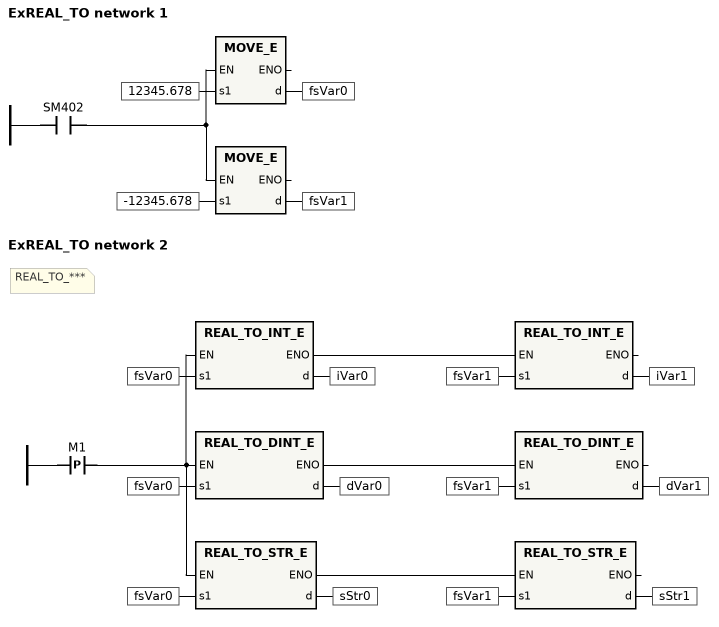
(* [picture p24: structured ladder/FBD of ExREAL_TO, networks 1 to 2] *)
(* network 1 *)
MOVE_E(SM402, 12345.678, fsVar0);
MOVE_E(SM402, -12345.678, fsVar1);
(* network 2 *)
(* REAL_TO_*** *)
_p1 := LDP(TRUE, M1);
_e2 := REAL_TO_INT_E(_p1, fsVar0, iVar0);
REAL_TO_INT_E(_e2, fsVar1, iVar1);
_e3 := REAL_TO_DINT_E(_p1, fsVar0, dVar0);
REAL_TO_DINT_E(_e3, fsVar1, dVar1);
_e4 := REAL_TO_STR_E(_p1, fsVar0, sStr0);
REAL_TO_STR_E(_e4, fsVar1, sStr1);
END_PROGRAM

PROGRAM ExSTR_TO
VAR
  GetInt : INT;
  NthBit : INT;
  SetInt : INT;
  SetInt2 : INT;
END_VAR
(* structured ladder/FBD written out as ST: instructions are called as NAME(EN, inputs, outputs); _pN, _eN, _tN stand for wires *)
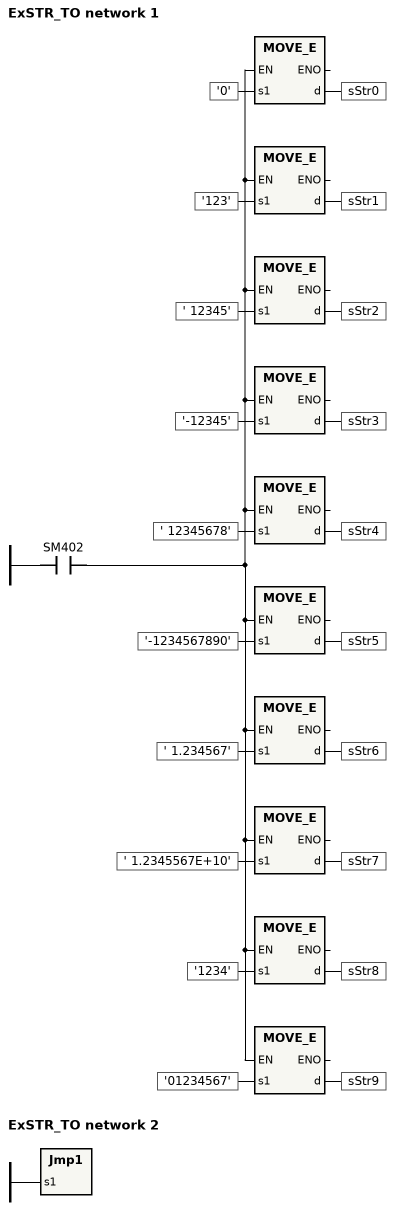
(* network 1 *)
MOVE_E(SM402, '0', sStr0);
MOVE_E(SM402, '123', sStr1);
MOVE_E(SM402, ' 12345', sStr2);
MOVE_E(SM402, '-12345', sStr3);
MOVE_E(SM402, ' 12345678', sStr4);
MOVE_E(SM402, '-1234567890', sStr5);
MOVE_E(SM402, ' 1.234567', sStr6);
MOVE_E(SM402, ' 1.2345567E+10', sStr7);
MOVE_E(SM402, '1234', sStr8);
MOVE_E(SM402, '01234567', sStr9);
(* network 2 *)
(* element kind 9 Jmp1 <- TRUE *)
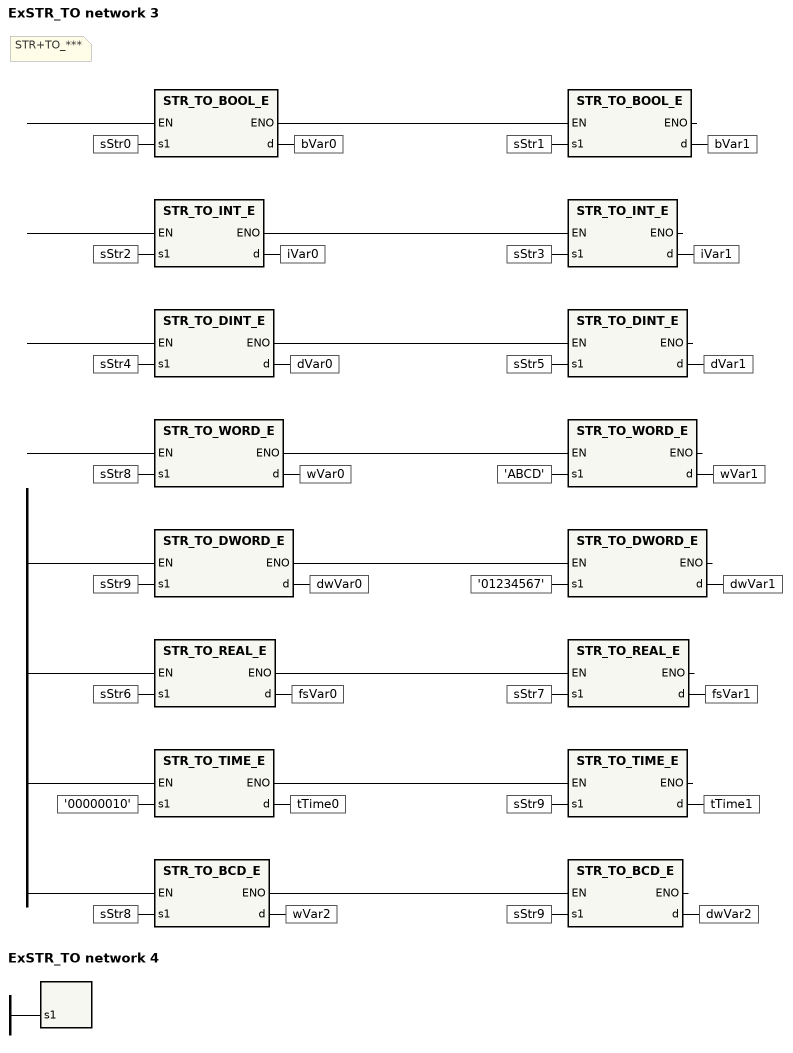
(* network 3 *)
(* STR+TO_*** *)
_e1 := STR_TO_BOOL_E(TRUE, sStr0, bVar0);
STR_TO_BOOL_E(_e1, sStr1, bVar1);
_e2 := STR_TO_INT_E(TRUE, sStr2, iVar0);
STR_TO_INT_E(_e2, sStr3, iVar1);
_e3 := STR_TO_DINT_E(TRUE, sStr4, dVar0);
STR_TO_DINT_E(_e3, sStr5, dVar1);
_e4 := STR_TO_WORD_E(TRUE, sStr8, wVar0);
STR_TO_WORD_E(_e4, 'ABCD', wVar1);
_e5 := STR_TO_DWORD_E(TRUE, sStr9, dwVar0);
STR_TO_DWORD_E(_e5, '01234567', dwVar1);
_e6 := STR_TO_REAL_E(TRUE, sStr6, fsVar0);
STR_TO_REAL_E(_e6, sStr7, fsVar1);
_e7 := STR_TO_TIME_E(TRUE, '00000010', tTime0);
STR_TO_TIME_E(_e7, sStr9, tTime1);
_e8 := STR_TO_BCD_E(TRUE, sStr8, wVar2);
STR_TO_BCD_E(_e8, sStr9, dwVar2);
(* network 4 *)
(* element kind 10  <- TRUE *)
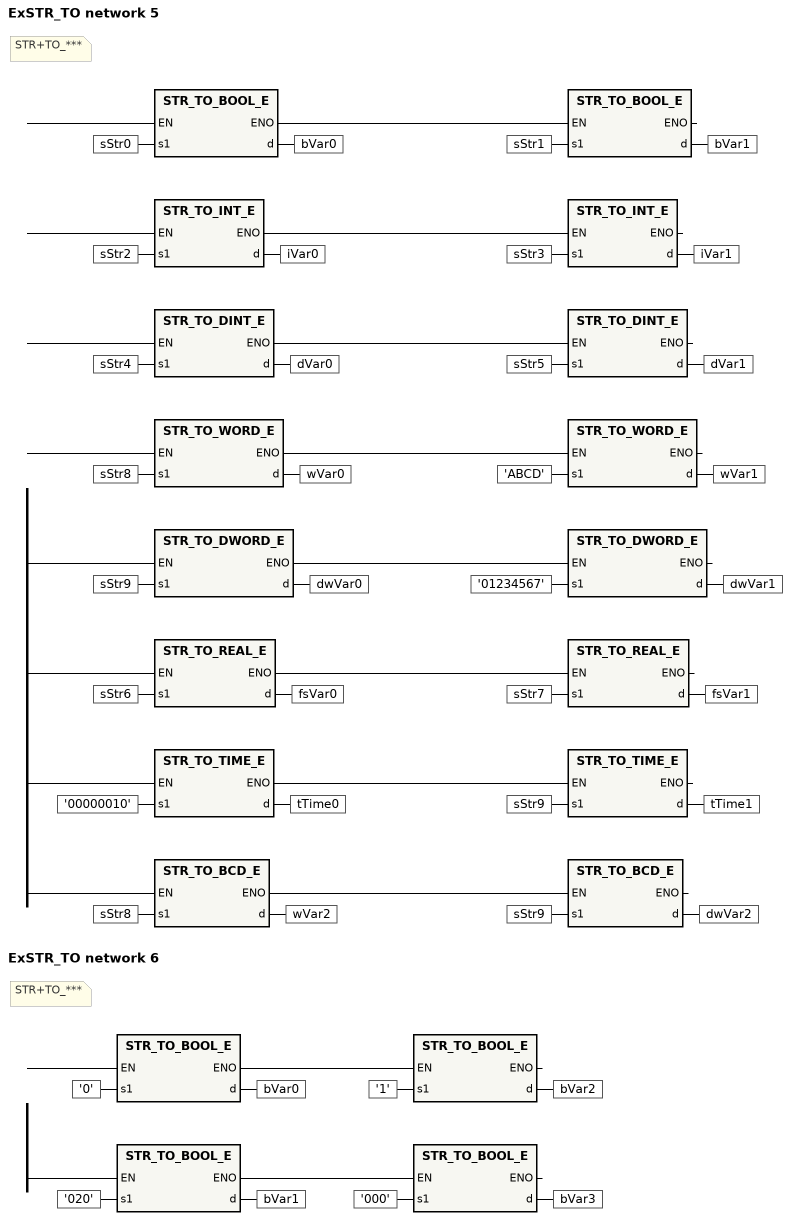
(* network 5 *)
(* STR+TO_*** *)
_e1 := STR_TO_BOOL_E(TRUE, sStr0, bVar0);
STR_TO_BOOL_E(_e1, sStr1, bVar1);
_e2 := STR_TO_INT_E(TRUE, sStr2, iVar0);
STR_TO_INT_E(_e2, sStr3, iVar1);
_e3 := STR_TO_DINT_E(TRUE, sStr4, dVar0);
STR_TO_DINT_E(_e3, sStr5, dVar1);
_e4 := STR_TO_WORD_E(TRUE, sStr8, wVar0);
STR_TO_WORD_E(_e4, 'ABCD', wVar1);
_e5 := STR_TO_DWORD_E(TRUE, sStr9, dwVar0);
STR_TO_DWORD_E(_e5, '01234567', dwVar1);
_e6 := STR_TO_REAL_E(TRUE, sStr6, fsVar0);
STR_TO_REAL_E(_e6, sStr7, fsVar1);
_e7 := STR_TO_TIME_E(TRUE, '00000010', tTime0);
STR_TO_TIME_E(_e7, sStr9, tTime1);
_e8 := STR_TO_BCD_E(TRUE, sStr8, wVar2);
STR_TO_BCD_E(_e8, sStr9, dwVar2);
(* network 6 Jmp1: *)
(* STR+TO_*** *)
_e1 := STR_TO_BOOL_E(TRUE, '0', bVar0);
STR_TO_BOOL_E(_e1, '1', bVar2);
_e2 := STR_TO_BOOL_E(TRUE, '020', bVar1);
STR_TO_BOOL_E(_e2, '000', bVar3);
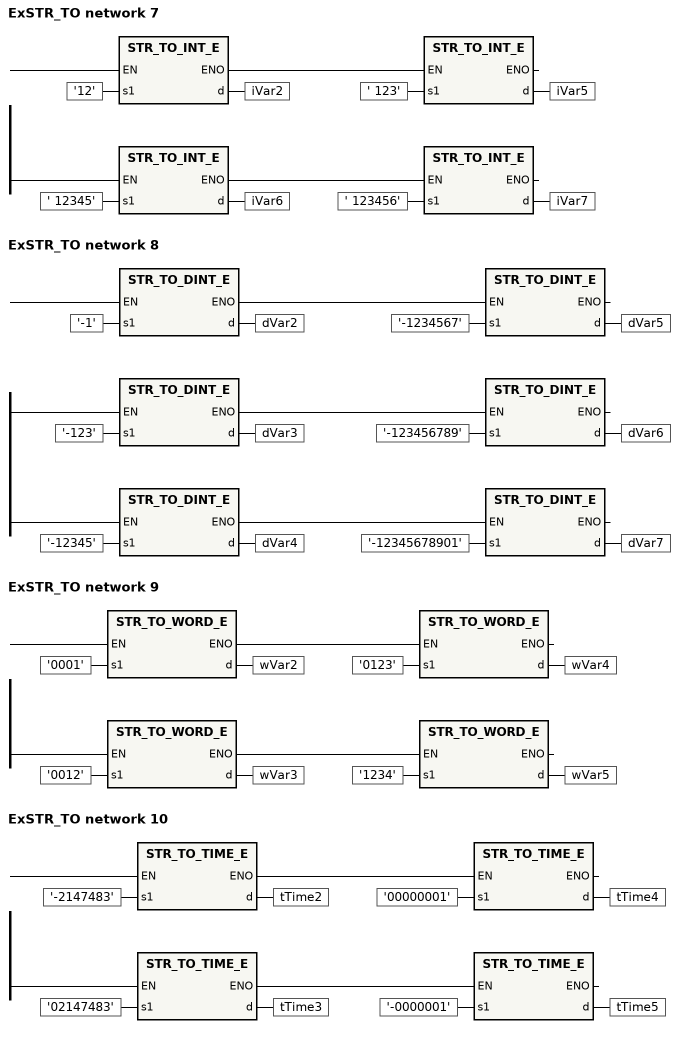
(* network 7 *)
_e1 := STR_TO_INT_E(TRUE, '12', iVar2);
STR_TO_INT_E(_e1, ' 123', iVar5);
_e2 := STR_TO_INT_E(TRUE, ' 12345', iVar6);
STR_TO_INT_E(_e2, ' 123456', iVar7);
(* network 8 *)
_e1 := STR_TO_DINT_E(TRUE, '-1', dVar2);
STR_TO_DINT_E(_e1, '-1234567', dVar5);
_e2 := STR_TO_DINT_E(TRUE, '-123', dVar3);
STR_TO_DINT_E(_e2, '-123456789', dVar6);
_e3 := STR_TO_DINT_E(TRUE, '-12345', dVar4);
STR_TO_DINT_E(_e3, '-12345678901', dVar7);
(* network 9 *)
_e1 := STR_TO_WORD_E(TRUE, '0001', wVar2);
STR_TO_WORD_E(_e1, '0123', wVar4);
_e2 := STR_TO_WORD_E(TRUE, '0012', wVar3);
STR_TO_WORD_E(_e2, '1234', wVar5);
(* network 10 *)
_e1 := STR_TO_TIME_E(TRUE, '-2147483', tTime2);
STR_TO_TIME_E(_e1, '00000001', tTime4);
_e2 := STR_TO_TIME_E(TRUE, '02147483', tTime3);
STR_TO_TIME_E(_e2, '-0000001', tTime5);
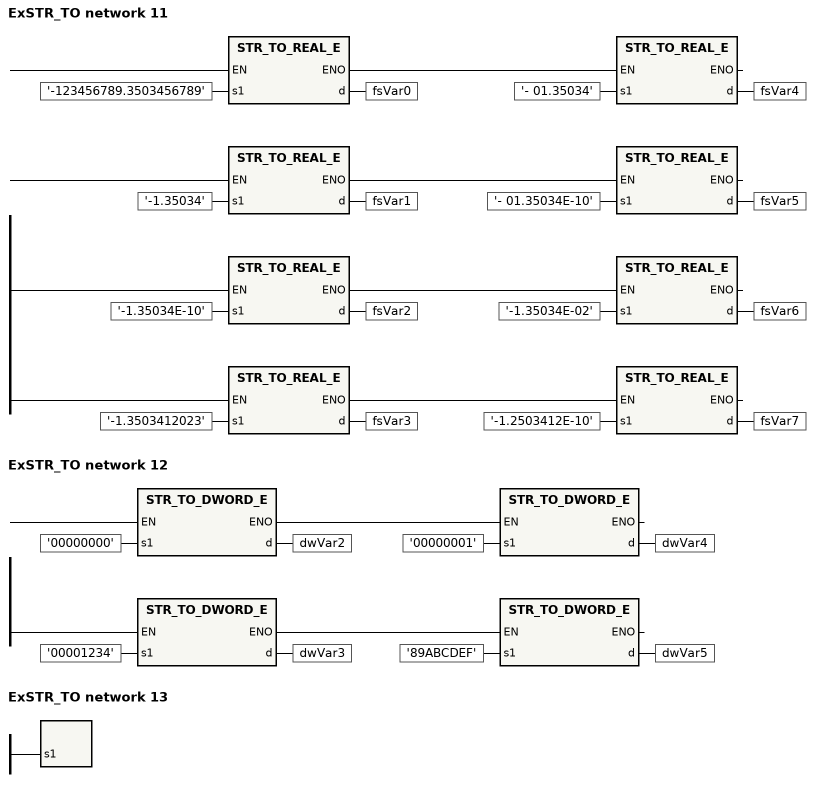
(* network 11 *)
_e1 := STR_TO_REAL_E(TRUE, '-123456789.3503456789', fsVar0);
STR_TO_REAL_E(_e1, '- 01.35034', fsVar4);
_e2 := STR_TO_REAL_E(TRUE, '-1.35034', fsVar1);
STR_TO_REAL_E(_e2, '- 01.35034E-10', fsVar5);
_e3 := STR_TO_REAL_E(TRUE, '-1.35034E-10', fsVar2);
STR_TO_REAL_E(_e3, '-1.35034E-02', fsVar6);
_e4 := STR_TO_REAL_E(TRUE, '-1.3503412023', fsVar3);
STR_TO_REAL_E(_e4, '-1.2503412E-10', fsVar7);
(* network 12 *)
_e1 := STR_TO_DWORD_E(TRUE, '00000000', dwVar2);
STR_TO_DWORD_E(_e1, '00000001', dwVar4);
_e2 := STR_TO_DWORD_E(TRUE, '00001234', dwVar3);
STR_TO_DWORD_E(_e2, '89ABCDEF', dwVar5);
(* network 13 *)
(* element kind 10  <- TRUE *)
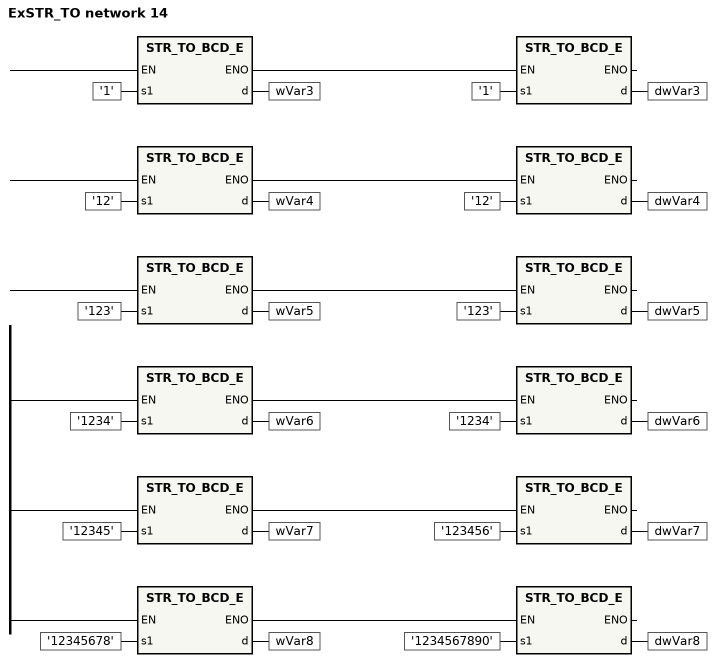
(* network 14 Jmp2: *)
_e1 := STR_TO_BCD_E(TRUE, '1', wVar3);
STR_TO_BCD_E(_e1, '1', dwVar3);
_e2 := STR_TO_BCD_E(TRUE, '12', wVar4);
STR_TO_BCD_E(_e2, '12', dwVar4);
_e3 := STR_TO_BCD_E(TRUE, '123', wVar5);
STR_TO_BCD_E(_e3, '123', dwVar5);
_e4 := STR_TO_BCD_E(TRUE, '1234', wVar6);
STR_TO_BCD_E(_e4, '1234', dwVar6);
_e5 := STR_TO_BCD_E(TRUE, '12345', wVar7);
STR_TO_BCD_E(_e5, '123456', dwVar7);
_e6 := STR_TO_BCD_E(TRUE, '12345678', wVar8);
STR_TO_BCD_E(_e6, '1234567890', dwVar8);
END_PROGRAM

PROGRAM ExTIME_TO
VAR
  GetInt : INT;
  NthBit : INT;
  SetInt : INT;
  SetInt2 : INT;
END_VAR
(* structured ladder/FBD written out as ST: instructions are called as NAME(EN, inputs, outputs); _pN, _eN, _tN stand for wires *)
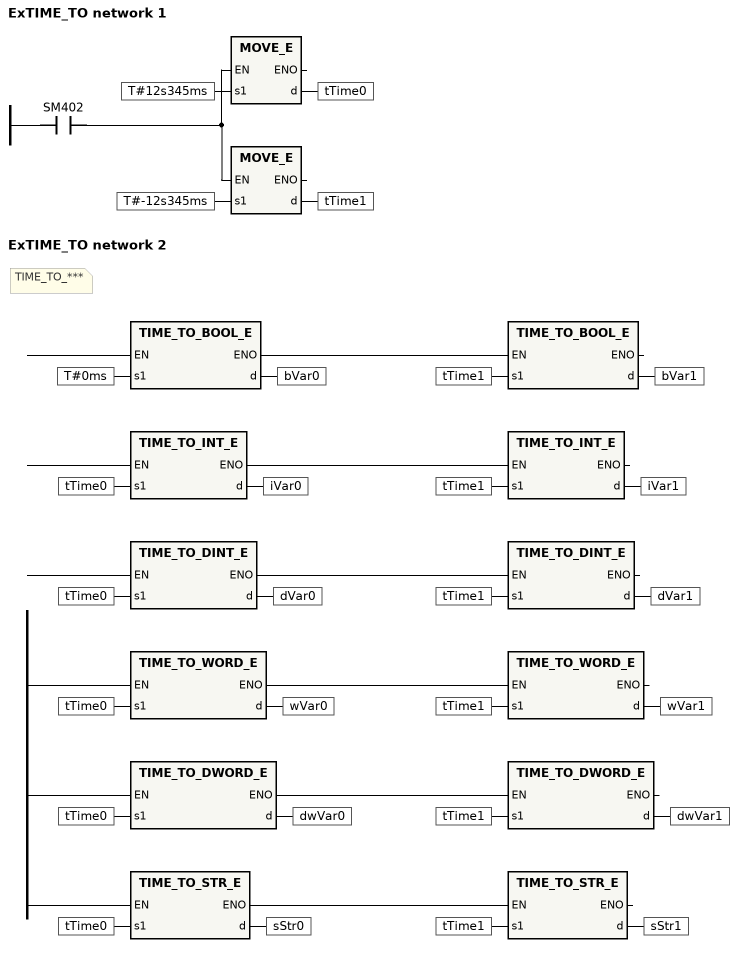
(* network 1 *)
MOVE_E(SM402, T#12s345ms, tTime0);
MOVE_E(SM402, T#-12s345ms, tTime1);
(* network 2 *)
(* TIME_TO_*** *)
_e1 := TIME_TO_BOOL_E(TRUE, T#0ms, bVar0);
TIME_TO_BOOL_E(_e1, tTime1, bVar1);
_e2 := TIME_TO_INT_E(TRUE, tTime0, iVar0);
TIME_TO_INT_E(_e2, tTime1, iVar1);
_e3 := TIME_TO_DINT_E(TRUE, tTime0, dVar0);
TIME_TO_DINT_E(_e3, tTime1, dVar1);
_e4 := TIME_TO_WORD_E(TRUE, tTime0, wVar0);
TIME_TO_WORD_E(_e4, tTime1, wVar1);
_e5 := TIME_TO_DWORD_E(TRUE, tTime0, dwVar0);
TIME_TO_DWORD_E(_e5, tTime1, dwVar1);
_e6 := TIME_TO_STR_E(TRUE, tTime0, sStr0);
TIME_TO_STR_E(_e6, tTime1, sStr1);
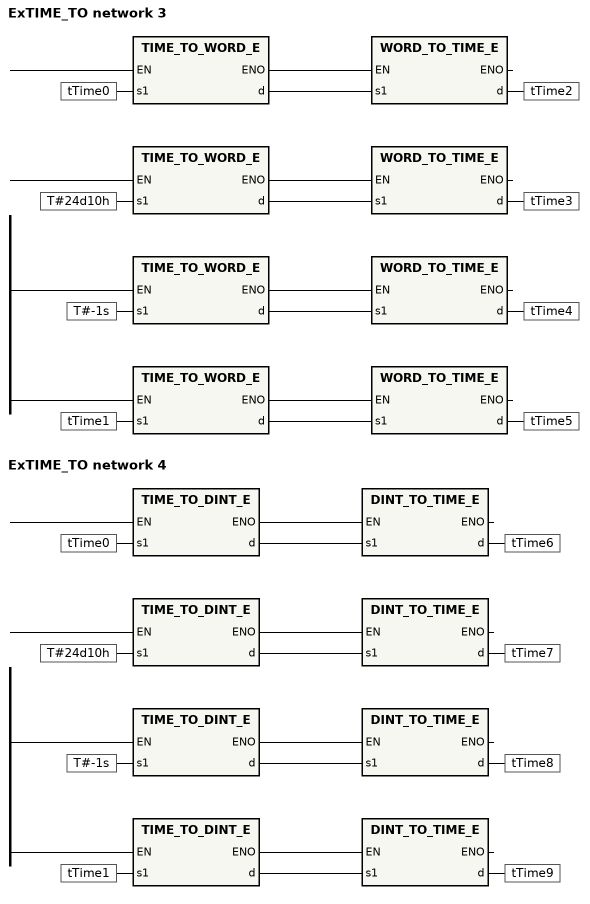
(* network 3 *)
_e2 := TIME_TO_WORD_E(TRUE, tTime0, _t1);
WORD_TO_TIME_E(_e2, _t1, tTime2);
_e4 := TIME_TO_WORD_E(TRUE, T#24d10h, _t3);
WORD_TO_TIME_E(_e4, _t3, tTime3);
_e6 := TIME_TO_WORD_E(TRUE, T#-1s, _t5);
WORD_TO_TIME_E(_e6, _t5, tTime4);
_e8 := TIME_TO_WORD_E(TRUE, tTime1, _t7);
WORD_TO_TIME_E(_e8, _t7, tTime5);
(* network 4 *)
_e2 := TIME_TO_DINT_E(TRUE, tTime0, _t1);
DINT_TO_TIME_E(_e2, _t1, tTime6);
_e4 := TIME_TO_DINT_E(TRUE, T#24d10h, _t3);
DINT_TO_TIME_E(_e4, _t3, tTime7);
_e6 := TIME_TO_DINT_E(TRUE, T#-1s, _t5);
DINT_TO_TIME_E(_e6, _t5, tTime8);
_e8 := TIME_TO_DINT_E(TRUE, tTime1, _t7);
DINT_TO_TIME_E(_e8, _t7, tTime9);
END_PROGRAM

PROGRAM ExWORD_TO
VAR
  GetInt : INT;
  NthBit : INT;
  SetInt : INT;
  SetInt2 : INT;
END_VAR
(* structured ladder/FBD written out as ST: instructions are called as NAME(EN, inputs, outputs); _pN, _eN, _tN stand for wires *)
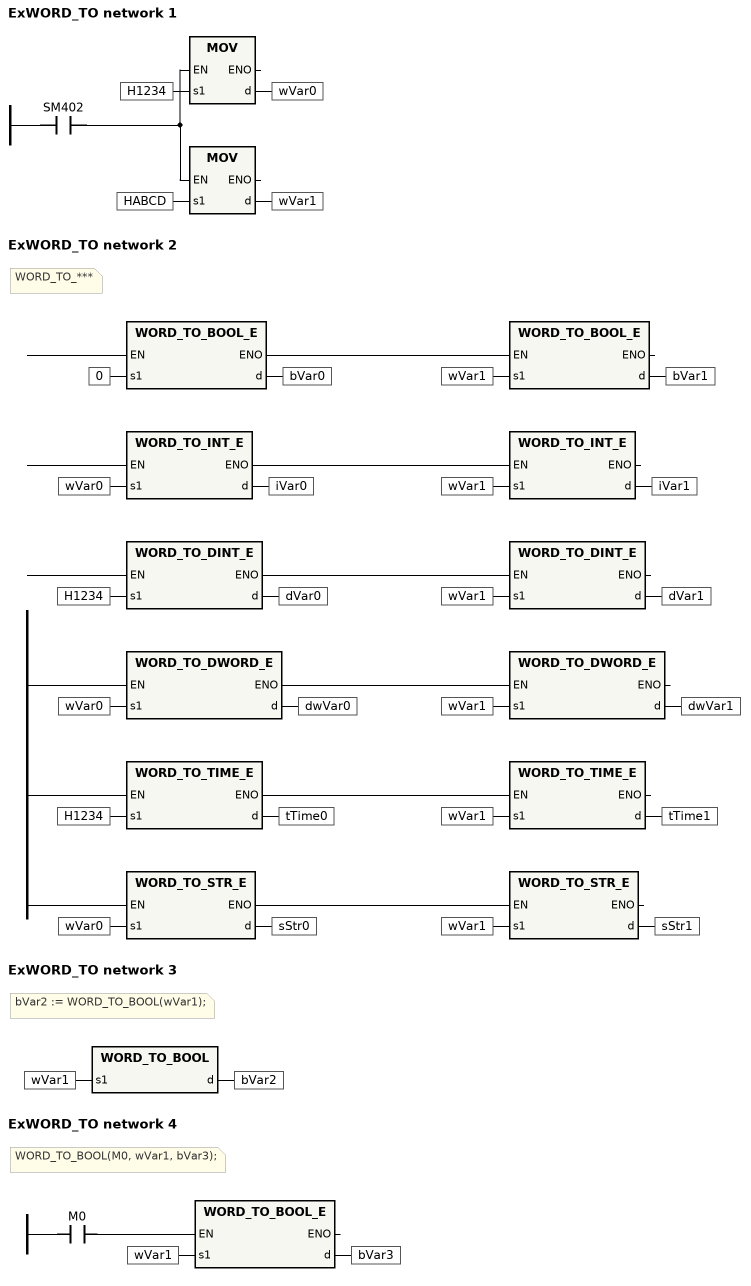
(* network 1 *)
MOV(SM402, H1234, wVar0);
MOV(SM402, HABCD, wVar1);
(* network 2 *)
(* WORD_TO_*** *)
_e1 := WORD_TO_BOOL_E(TRUE, 0, bVar0);
WORD_TO_BOOL_E(_e1, wVar1, bVar1);
_e2 := WORD_TO_INT_E(TRUE, wVar0, iVar0);
WORD_TO_INT_E(_e2, wVar1, iVar1);
_e3 := WORD_TO_DINT_E(TRUE, H1234, dVar0);
WORD_TO_DINT_E(_e3, wVar1, dVar1);
_e4 := WORD_TO_DWORD_E(TRUE, wVar0, dwVar0);
WORD_TO_DWORD_E(_e4, wVar1, dwVar1);
_e5 := WORD_TO_TIME_E(TRUE, H1234, tTime0);
WORD_TO_TIME_E(_e5, wVar1, tTime1);
_e6 := WORD_TO_STR_E(TRUE, wVar0, sStr0);
WORD_TO_STR_E(_e6, wVar1, sStr1);
(* network 3 *)
(* bVar2 := WORD_TO_BOOL(wVar1); *)
bVar2 := WORD_TO_BOOL(wVar1);
(* network 4 *)
(* WORD_TO_BOOL(M0, wVar1, bVar3); *)
WORD_TO_BOOL_E(M0, wVar1, bVar3);
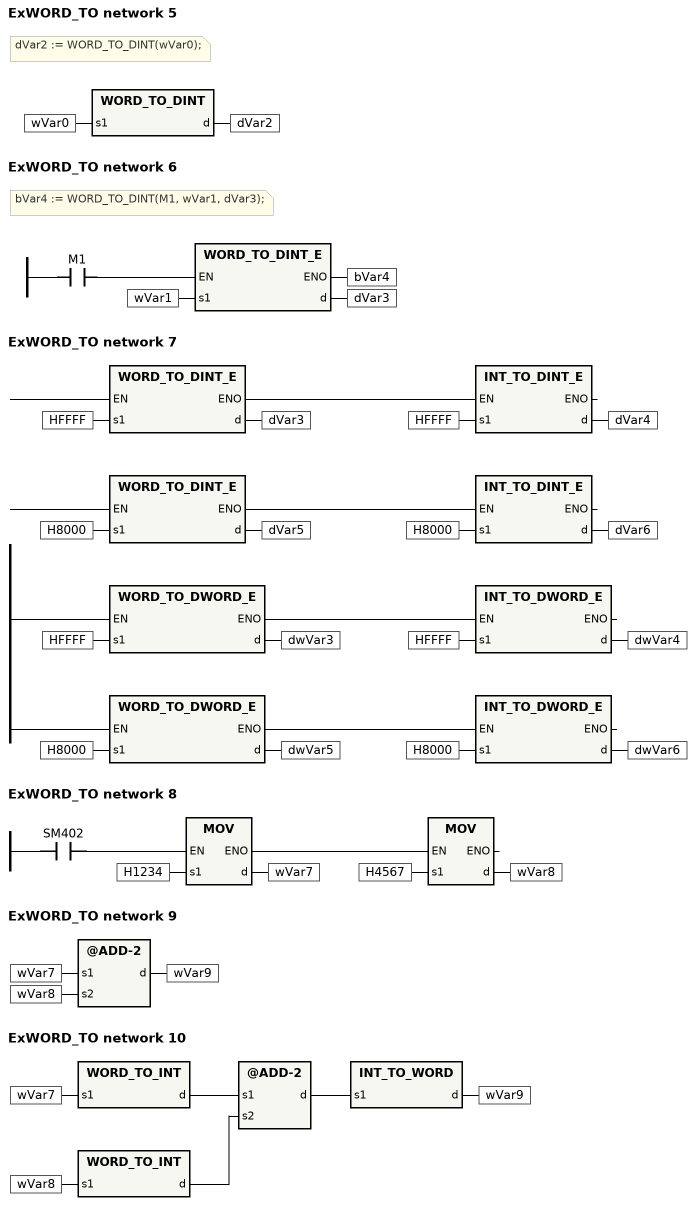
(* network 5 *)
(* dVar2 := WORD_TO_DINT(wVar0); *)
dVar2 := WORD_TO_DINT(wVar0);
(* network 6 *)
(* bVar4 := WORD_TO_DINT(M1, wVar1, dVar3); *)
_e1 := WORD_TO_DINT_E(M1, wVar1, dVar3);
bVar4 := _e1;
(* network 7 *)
_e1 := WORD_TO_DINT_E(TRUE, HFFFF, dVar3);
INT_TO_DINT_E(_e1, HFFFF, dVar4);
_e2 := WORD_TO_DINT_E(TRUE, H8000, dVar5);
INT_TO_DINT_E(_e2, H8000, dVar6);
_e3 := WORD_TO_DWORD_E(TRUE, HFFFF, dwVar3);
INT_TO_DWORD_E(_e3, HFFFF, dwVar4);
_e4 := WORD_TO_DWORD_E(TRUE, H8000, dwVar5);
INT_TO_DWORD_E(_e4, H8000, dwVar6);
(* network 8 *)
_e1 := MOV(SM402, H1234, wVar7);
MOV(_e1, H4567, wVar8);
(* network 9 *)
wVar9 := @ADD-2(wVar7, wVar8);
(* network 10 *)
wVar9 := INT_TO_WORD(@ADD-2(WORD_TO_INT(wVar7), WORD_TO_INT(wVar8)));
END_PROGRAM

FUNCTION_BLOCK INT2Bit
VAR_INPUT
  IN : INT;
END_VAR
VAR_OUTPUT
  Bit0 : BOOL;
  Bit1 : BOOL;
  Bit2 : BOOL;
  Bit3 : BOOL;
  Bit4 : BOOL;
  Bit5 : BOOL;
  Bit6 : BOOL;
  Bit7 : BOOL;
  Bit8 : BOOL;
  Bit9 : BOOL;
  Bit10 : BOOL;
  Bit11 : BOOL;
  Bit12 : BOOL;
  Bit13 : BOOL;
  Bit14 : BOOL;
  Bit15 : BOOL;
END_VAR
VAR
  abArr16 : ARRAY [0..15] OF BOOL;
END_VAR
 
abArr16[0] := INT_TO_BITARR(IN, 16);
Bit0 := abArr16[0];
Bit1 := abArr16[1];
Bit2 := abArr16[2];
Bit3 := abArr16[3];
Bit4 := abArr16[4];
Bit5 := abArr16[5];
Bit6 := abArr16[6];
Bit7 := abArr16[7];
Bit8 := abArr16[8];
Bit9 := abArr16[9];
Bit10 := abArr16[10];
Bit11 := abArr16[11];
Bit12 := abArr16[12];
Bit13 := abArr16[13];
Bit14 := abArr16[14];
Bit15 := abArr16[15];
END_FUNCTION_BLOCK

PROGRAM ExBCD_TO2
VAR
  aTank : ARRAY [0..31] OF INT;
  awStatus : ARRAY [0..9] OF WORD;
  asName : ARRAY [0..4] OF STRING[32] := [5('')];
  atDelay : ARRAY [0..4] OF TIME := [5(T#0s)];
  HMI20_1 : HMI20;
  Mov4WORD_1 : Mov4WORD;
  Mov4DWORD_1 : Mov4DWORD;
END_VAR
(* structured ladder/FBD written out as ST: instructions are called as NAME(EN, inputs, outputs); _pN, _eN, _tN stand for wires *)
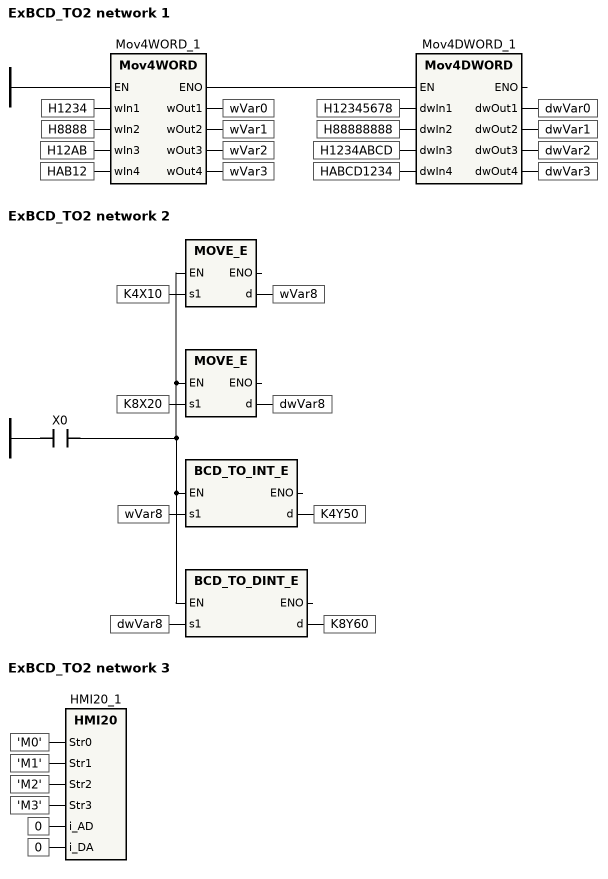
(* network 1 *)
Mov4WORD_1(EN := TRUE, wIn1 := H1234, wIn2 := H8888, wIn3 := H12AB, wIn4 := HAB12, wOut1 => wVar0, wOut2 => wVar1, wOut3 => wVar2, wOut4 => wVar3);
Mov4DWORD_1(EN := Mov4WORD_1.ENO, dwIn1 := H12345678, dwIn2 := H88888888, dwIn3 := H1234ABCD, dwIn4 := HABCD1234, dwOut1 => dwVar0, dwOut2 => dwVar1, dwOut3 => dwVar2, dwOut4 => dwVar3);
(* network 2 *)
MOVE_E(X0, K4X10, wVar8);
MOVE_E(X0, K8X20, dwVar8);
BCD_TO_INT_E(X0, wVar8, K4Y50);
BCD_TO_DINT_E(X0, dwVar8, K8Y60);
(* network 3 *)
HMI20_1(Str0 := 'M0', Str1 := 'M1', Str2 := 'M2', Str3 := 'M3', i_AD := 0, i_DA := 0);
END_PROGRAM

PROGRAM ExBCD_TO
VAR
  aTank : ARRAY [0..31] OF INT;
  awStatus : ARRAY [0..9] OF WORD;
  asName : ARRAY [0..4] OF STRING[32] := [5('')];
  atDelay : ARRAY [0..4] OF TIME := [5(T#0s)];
  HMI20_1 : HMI20;
  Mov4WORD_1 : Mov4WORD;
  Mov4DWORD_1 : Mov4DWORD;
END_VAR
(* structured ladder/FBD written out as ST: instructions are called as NAME(EN, inputs, outputs); _pN, _eN, _tN stand for wires *)
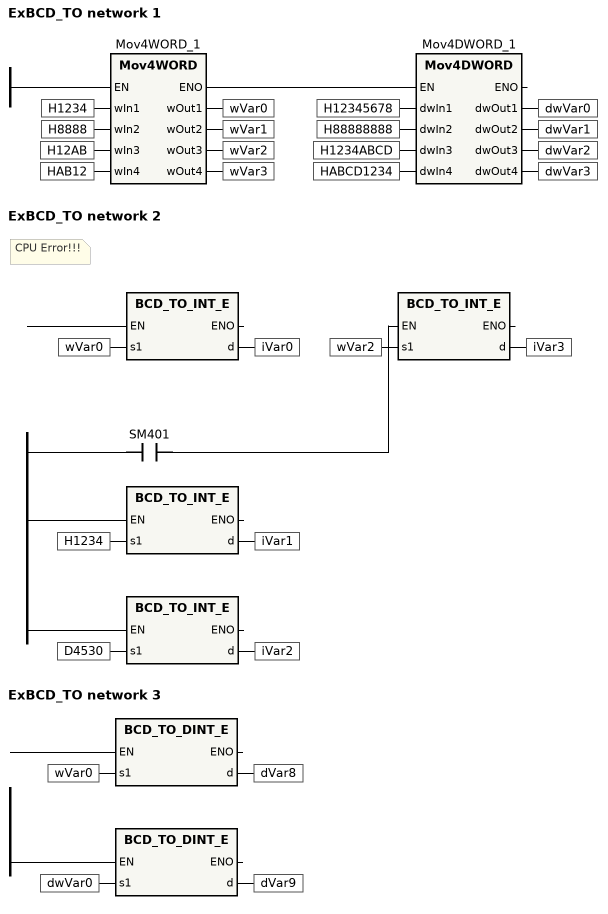
(* network 1 *)
Mov4WORD_1(EN := TRUE, wIn1 := H1234, wIn2 := H8888, wIn3 := H12AB, wIn4 := HAB12, wOut1 => wVar0, wOut2 => wVar1, wOut3 => wVar2, wOut4 => wVar3);
Mov4DWORD_1(EN := Mov4WORD_1.ENO, dwIn1 := H12345678, dwIn2 := H88888888, dwIn3 := H1234ABCD, dwIn4 := HABCD1234, dwOut1 => dwVar0, dwOut2 => dwVar1, dwOut3 => dwVar2, dwOut4 => dwVar3);
(* network 2 *)
(* CPU Error!!! *)
BCD_TO_INT_E(TRUE, wVar0, iVar0);
BCD_TO_INT_E(TRUE, H1234, iVar1);
BCD_TO_INT_E(TRUE, D4530, iVar2);
BCD_TO_INT_E(SM401, wVar2, iVar3);
(* network 3 *)
BCD_TO_DINT_E(TRUE, wVar0, dVar8);
BCD_TO_DINT_E(TRUE, dwVar0, dVar9);
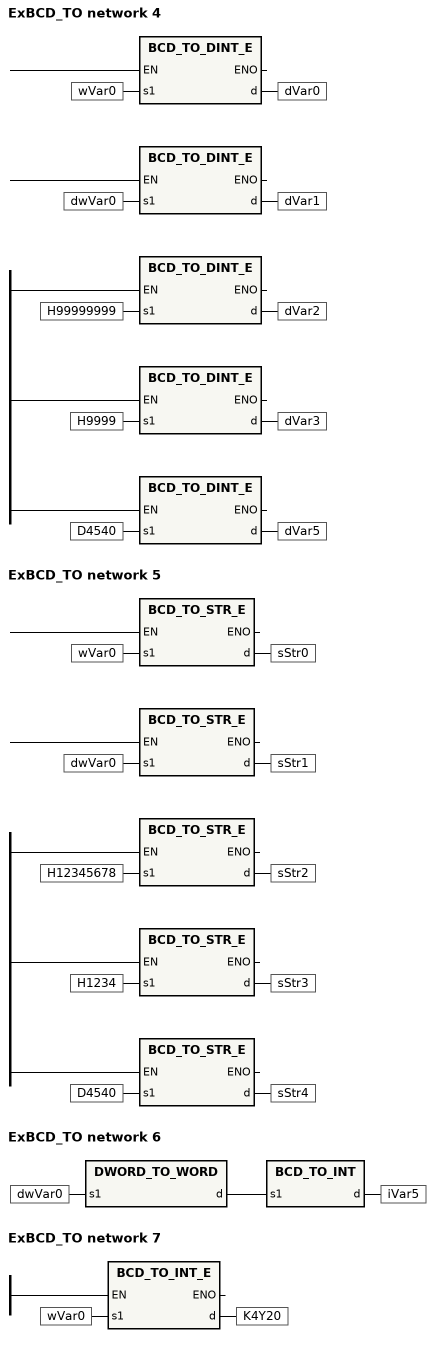
(* network 4 *)
BCD_TO_DINT_E(TRUE, wVar0, dVar0);
BCD_TO_DINT_E(TRUE, dwVar0, dVar1);
BCD_TO_DINT_E(TRUE, H99999999, dVar2);
BCD_TO_DINT_E(TRUE, H9999, dVar3);
BCD_TO_DINT_E(TRUE, D4540, dVar5);
(* network 5 *)
BCD_TO_STR_E(TRUE, wVar0, sStr0);
BCD_TO_STR_E(TRUE, dwVar0, sStr1);
BCD_TO_STR_E(TRUE, H12345678, sStr2);
BCD_TO_STR_E(TRUE, H1234, sStr3);
BCD_TO_STR_E(TRUE, D4540, sStr4);
(* network 6 *)
iVar5 := BCD_TO_INT(DWORD_TO_WORD(dwVar0));
(* network 7 *)
BCD_TO_INT_E(TRUE, wVar0, K4Y20);
END_PROGRAM

FUNCTION Word2Dint
VAR_INPUT
  LoW : WORD;
  HiW : WORD;
END_VAR
VAR
  dwMergeL : DWORD;
  dwMergeH : DWORD;
  dwMerge : DWORD;
END_VAR
;
dwMergeL 	:= WORD_TO_DWORD(LoW);
dwMergeH 	:= WORD_TO_DWORD(HiW);
dwMerge 		:= SHL(dwMergeH , 16) OR dwMergeL;
Word2Dint 	:= DWORD_TO_DINT(dwMerge);
END_FUNCTION

FUNCTION_BLOCK Dint2Word
VAR_INPUT
  dDINT : DINT;
END_VAR
VAR_OUTPUT
  wLO : WORD;
  wHI : WORD;
END_VAR
VAR
  dwTemp : DWORD;
END_VAR
;
dwTemp	:= DINT_TO_DWORD(dDINT);
wLO			:= DWORD_TO_WORD(dwTemp AND HFFFF);
wHI				:= DWORD_TO_WORD(SHR(dwTemp , 16) AND HFFFF);
END_FUNCTION_BLOCK

PROGRAM ExWORD2DINT
VAR
  Mov4WORD_1 : Mov4WORD;
END_VAR
(* structured ladder/FBD written out as ST: instructions are called as NAME(EN, inputs, outputs); _pN, _eN, _tN stand for wires *)
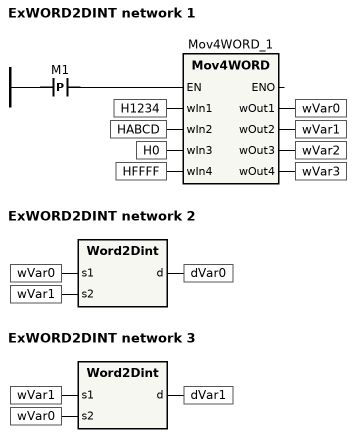
(* network 1 *)
Mov4WORD_1(EN := LDP(TRUE, M1), wIn1 := H1234, wIn2 := HABCD, wIn3 := H0, wIn4 := HFFFF, wOut1 => wVar0, wOut2 => wVar1, wOut3 => wVar2, wOut4 => wVar3);
(* network 2 *)
dVar0 := Word2Dint(wVar0, wVar1);
(* network 3 *)
dVar1 := Word2Dint(wVar1, wVar0);
END_PROGRAM

PROGRAM ExDINT2WORD
VAR
  Dint2Word_1 : Dint2Word;
  Dint2Word_2 : Dint2Word;
  Dint2Word_3 : Dint2Word;
END_VAR
(* structured ladder/FBD written out as ST: instructions are called as NAME(EN, inputs, outputs); _pN, _eN, _tN stand for wires *)
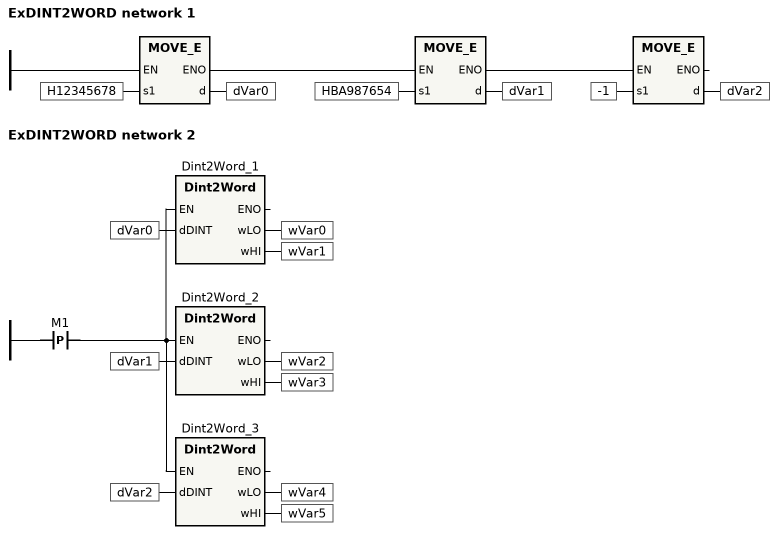
(* network 1 *)
_e1 := MOVE_E(TRUE, H12345678, dVar0);
_e2 := MOVE_E(_e1, HBA987654, dVar1);
MOVE_E(_e2, -1, dVar2);
(* network 2 *)
_p1 := LDP(TRUE, M1);
Dint2Word_1(EN := _p1, dDINT := dVar0, wLO => wVar0, wHI => wVar1);
Dint2Word_2(EN := _p1, dDINT := dVar1, wLO => wVar2, wHI => wVar3);
Dint2Word_3(EN := _p1, dDINT := dVar2, wLO => wVar4, wHI => wVar5);
END_PROGRAM
